{attribute 'qualified_only'}
VAR_GLOBAL
	upperDistance 	: 	INT 	:= 10;
	lowerDistance	: 	INT 	:= 1;
	counter3	:	INT		:= 69;	
END_VAR

(* stored: Version 1.1.0.1, ProductVersion 3.1.4024.10
   GVL AdsVariables: Id {186c5690-a863-4347-bace-605c9d8bf706} *)
